Staubli VAL3: remCalcHere.pgx

program remCalcHere()
  local point pHere
  local trsf trHere
begin
  // Calculate current position in current frame and save to globals
  //
  logMsg("call remCalcHere")
  if nIPNumber==0
    pHere=here(tSensorTool,fIP1)
  else
    pHere=here(tSensorTool,fIP2)
  endIf
  trHere=pHere.trsf
  nXHere=trHere.x
  nYHere=trHere.y
  nZHere=trHere.z
  nRXHere=trHere.rx
  nRYHere=trHere.ry
  nRZHere=trHere.rz
end
